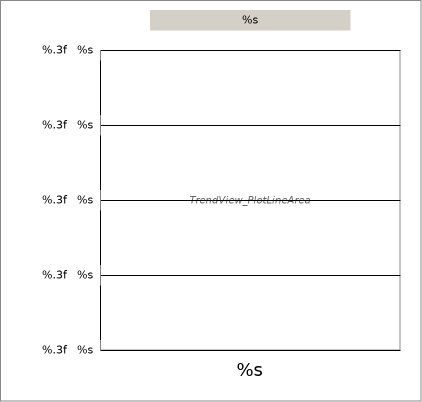
VISUALIZATION TrendView  // 422x402
VAR_IN_OUT
	PLC_IN : M_TRENDVIEW_OBJECT;
END_VAR
    Rectangle (0,0 420x400)
    Frame (100,50 300x300)
        shows TrendView_PlotLineArea(PLC_IN := PLC_IN)
    Line (100,50) (100,350)
    Line (100,350) (400,350)
    Line (100,200) (400,200)
    Line (100,125) (400,125)
    Line (100,275) (400,275)
    Line (100,50) (400,50)
    Textfield (20,40 50x20), "%.3f", text variable: PLC_IN.AXIS_Y_MAX, input disabled if: TRUE
    Textfield (70,40 30x20), "%s", text variable: PLC_IN.DISPLAY_Y_UNIT, input disabled if: TRUE
    Textfield (20,340 50x20), "%.3f", text variable: PLC_IN.AXIS_Y_MIN, input disabled if: TRUE
    Textfield (70,340 30x20), "%s", text variable: PLC_IN.DISPLAY_Y_UNIT, input disabled if: TRUE
    Textfield (200,360 100x20), "%s", text variable: PLC_IN.DISPLAY_X_AXIS_LABEL, input disabled if: TRUE
    Textfield (20,115 50x20), "%.3f", text variable: ((PLC_IN.AXIS_Y_MAX - PLC_IN.AXIS_Y_MIN) * 0.75) + PLC_IN.AXIS_Y_MIN, input disabled if: TRUE
    Textfield (70,115 30x20), "%s", text variable: PLC_IN.DISPLAY_Y_UNIT, input disabled if: TRUE
    Textfield (20,190 50x20), "%.3f", text variable: ((PLC_IN.AXIS_Y_MAX - PLC_IN.AXIS_Y_MIN) * 0.5) + PLC_IN.AXIS_Y_MIN, input disabled if: TRUE
    Textfield (70,190 30x20), "%s", text variable: PLC_IN.DISPLAY_Y_UNIT, input disabled if: TRUE
    Textfield (20,265 50x20), "%.3f", text variable: ((PLC_IN.AXIS_Y_MAX - PLC_IN.AXIS_Y_MIN) * 0.25) + PLC_IN.AXIS_Y_MIN, input disabled if: TRUE
    Textfield (70,265 30x20), "%s", text variable: PLC_IN.DISPLAY_Y_UNIT, input disabled if: TRUE
    Textfield (150,10 200x20), "%s", text variable: PLC_IN.DISPLAY_TITLE
END_VISUALIZATION

(* stored: Version 1.1.0.1, ProductVersion 3.1.4020.3
   Visu TrendView: Id {b169edcf-758b-4948-9abd-87005bb4d643} *)
